{attribute 'qualified_only'}
{attribute 'strict'}
TYPE E_Vise_Command :
(
	Load,
	InProcess,
	UnLoad
);
END_TYPE

(* stored: Version 1.1.0.1, ProductVersion 3.1.4024.11
   DUT E_Vise_Command: Id {f6f4a53f-dffe-4fb8-8804-bd2b59577fb2} *)
